FUNCTION F_ClearError 
VAR_INPUT
	Error : REFERENCE TO ST_Error;
END_VAR
VAR
END_VAR

IF __ISVALIDREF(Error) THEN 
	Error.Active := FALSE;
	Error.Label := '';
	Error.Message := '';
	Error.Priority := E_ErrorPriority.Diagnostic;
END_IF

END_FUNCTION

(* stored: Version 1.1.0.1, ProductVersion 3.1.4024.12
   POU F_ClearError: Id {a8ff4cbd-6e27-46d1-854a-76e8fce49f6b}, SpecialFunc None *)
